{attribute 'linkalways'} 
{attribute 'no_explicit_call' := 'This FB is a CLASS and must be accessed using methods or properties'}
{attribute 'enable_dynamic_creation'}
FUNCTION_BLOCK FINAL GE_REAL EXTENDS Node
VAR
	in1 : _REAL(0.0);
	in2 : _REAL(0.0);
	out : _BOOL(FALSE);
END_VAR

METHOD PUBLIC Clone : I_Node
VAR
	pNode : POINTER TO GE_REAL;
END_VAR
pNode := __NEW(GE_REAL);
Clone := pNode^;
END_METHOD

METHOD FB_init : BOOL
VAR_INPUT
	bInitRetains : BOOL; // if TRUE, the retain variables are initialized (warm start / cold start)
	bInCopyCode : BOOL;  // if TRUE, the instance afterwards gets moved into the copy code (online change)
END_VAR
AddInput('in1',THIS^.in1);
AddInput('in2',THIS^.in2);
AddOutput('out', THIS^.out);
END_METHOD

METHOD PROTECTED OnExecute
VAR
END_VAR
out.Value := in1.Value >= in2.Value;
END_METHOD

END_FUNCTION_BLOCK

(* stored: Version 1.1.0.1, ProductVersion 3.1.4024.15
   POU GE_REAL: Id {608aa5a6-756b-4dff-920d-44e3f81986dc}, SpecialFunc None
   Folder Constructor: Id {ee9acd69-b390-457b-a15c-88526740bba1}
   Method Clone: Id {d8efc008-dd12-45b7-b2aa-afa44c17dbab}
   Method FB_init: Id {719fe7e5-cebb-4efd-90c6-44a50f1b5773}
   Method OnExecute: Id {51f31001-37b6-4ff7-97f3-c71b433e9dae} *)
